SUBAPPLICATION Uebung_020i (* DigitalInput_I1 auf DigitalOutput_Q1; E_PULSE; Impulsformend; Teach-In *)
  (* Standard: 61499-2; Description: Copyright (c) 2023 Meisterschulen am Ostbahnhof This program and the accompanying materials are made available under the terms of the Eclipse Public License 2.0 which is available at https://www.eclipse.org/legal/epl-2.0/ SPDX-License-Identifier: EPL-2.0 *)
  (* Version 1.0, 2023-10-23, Franz Höpfinger, Meisterschulen am Ostbahnhof *)
  PACKAGE Uebungen;
  IMPORT logiBUS::io::DI::logiBUS_DI::Input_I1;
  IMPORT logiBUS::io::DI::logiBUS_DI::Input_I2;
  IMPORT logiBUS::io::DI::logiBUS_DI_Events::BUTTON_SINGLE_CLICK;
  IMPORT logiBUS::io::DQ::logiBUS_DO::Output_Q1;
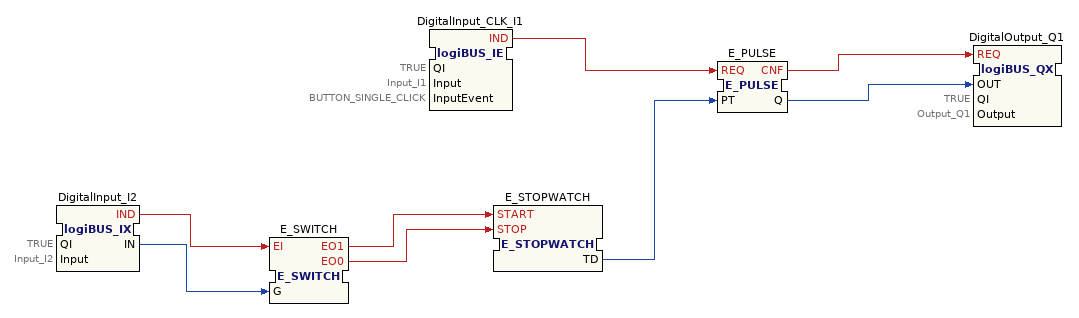
  FBS
    DigitalOutput_Q1 : logiBUS::io::DQ::logiBUS_QX(QI := TRUE, Output := Output_Q1);
    E_PULSE : iec61499::events::timers::E_PULSE;
    DigitalInput_CLK_I1 : logiBUS::io::DI::logiBUS_IE(QI := TRUE, Input := Input_I1, InputEvent := BUTTON_SINGLE_CLICK);
    E_STOPWATCH : eclipse4diac::utils::timing::E_STOPWATCH;
    E_SWITCH : iec61499::events::E_SWITCH;
    DigitalInput_I2 : logiBUS::io::DI::logiBUS_IX(QI := TRUE, Input := Input_I2);
  END_FBS
  EVENT_CONNECTIONS
    E_PULSE.CNF TO DigitalOutput_Q1.REQ;
    DigitalInput_CLK_I1.IND TO E_PULSE.REQ;
    DigitalInput_I2.IND TO E_SWITCH.EI;
    E_SWITCH.EO1 TO E_STOPWATCH.START;
    E_SWITCH.EO0 TO E_STOPWATCH.STOP;
  END_CONNECTIONS
  DATA_CONNECTIONS
    E_PULSE.Q TO DigitalOutput_Q1.OUT;
    E_STOPWATCH.TD TO E_PULSE.PT;
    DigitalInput_I2.IN TO E_SWITCH.G;
  END_CONNECTIONS
END_SUBAPPLICATION
